// TwinCAT 3 PLC project PLC
// Title: AUT_Utilities
// Company: AU-tomation
// Author: Ing. Alberto Utili
// ProjectVersion: 1.0.0.0
// Description: AU-tomation Toolkit Utilities Library
// ProgramVersion: 3.1.4026.20
// libraries:
//   Tc2_Standard, * (Beckhoff Automation GmbH)
//   Tc2_System, * (Beckhoff Automation GmbH)
//   Tc2_Utilities, * (Beckhoff Automation GmbH)
//   Tc3_Module, * (Beckhoff Automation GmbH)
// project tree:
//   POUs/StringBuilder/Classes/ StringBuilder.TcPOU
//   POUs/StringBuilder/Interfaces/ ILimitedStringBuilder.TcIO, IStringBuilder.TcIO (not stored)
//   Project Information/ F_GetCompany.TcPOU, F_GetTitle.TcPOU, F_GetVersion.TcPOU
//   Version/ Global_Version.TcGVL

// ---- Version/Global_Version.TcGVL
{attribute 'TcGenerated'}
{attribute 'no-analysis'}
{attribute 'linkalways'}
// This function has been automatically generated from the project information.
VAR_GLOBAL CONSTANT
	{attribute 'const_non_replaced'}
	stLibVersion_AUT_Utilities : ST_LibVersion := (iMajor := 1, iMinor := 0, iBuild := 0, iRevision := 0, nFlags := 0, sVersion := '1.0.0.0');
END_VAR

// ---- POUs/StringBuilder/Interfaces/ILimitedStringBuilder.TcIO
INTERFACE ILimitedStringBuilder

METHOD  Append : IStringBuilder // Append text to t current build string.
VAR_INPUT
	Text : STRING(1024); //Text to append to current build string
END_VAR
END_METHOD

METHOD Reset : ILimitedStringBuilder //Reset current build string to an empty string.
END_METHOD

METHOD ToString : STRING(2048)    //Returns current build string.
END_METHOD

METHOD ToWString : WSTRING(2048) //Returns current build string.
END_METHOD

END_INTERFACE

// ---- POUs/StringBuilder/Classes/StringBuilder.TcPOU
FUNCTION_BLOCK PUBLIC StringBuilder IMPLEMENTS  IStringBuilder, ILimitedStringBuilder
VAR
	{attribute 'hide'}
	_BuildingString : STRING(2048);
END_VAR

METHOD PUBLIC Append : IStringBuilder // Append text to t current build string.
VAR_INPUT
	Text : STRING(1024); //Text to append to current build string
END_VAR
VAR
    _BoolRes : BOOL;
END_VAR
_BoolRes := Tc2_Utilities.CONCAT2(ADR(_BuildingString), ADR(Text), ADR(_BuildingString), SIZEOF(_BuildingString));
Append := THIS^;    // Fluent interface
END_METHOD

METHOD AssignDelimitedSubstringTo : IStringBuilder
VAR_INPUT
    Delimiter : STRING(1);
    SubstringIndex : UDINT;
	Destination : POINTER TO STRING(2048);
    DestinationSize : UDINT;
END_VAR
VAR
    _CurrentPosition : UDINT := 0;
    _CurrentDelimiterPosition : UDINT := 0;
    _CurrentDelimiterIndex : UDINT := 0;
    _LeadingDelimiterPosition : UDINT := 0;
    _TrailingDelimiterPosition : UDINT := 0;
    _Substring : STRING(2048) := '';
    _Index : UDINT;
    _BoolRes : BOOL;
END_VAR
// FOR _Index := 1 TO (SubstringIndex - 1) DO
//     _LeadingDelimiterPosition := Tc2_Utilities.FIND2(ADR(_BuildingString), ADR(Delimiter))
//     
// END_FOR

// ATTENTION: pointer arithmetics is used to move inside string
IF SubstringIndex < 1 THEN
    SubstringIndex := 1;
END_IF
REPEAT
    _CurrentDelimiterPosition := Tc2_Utilities.FIND2(ADR(_BuildingString) + _CurrentPosition, ADR(Delimiter));
    IF _CurrentDelimiterPosition > 0 THEN
        _CurrentPosition := _CurrentPosition + _CurrentDelimiterPosition;
        _CurrentDelimiterIndex := _CurrentDelimiterIndex + 1;
        IF _CurrentDelimiterIndex = (SubstringIndex - 1) THEN
            _LeadingDelimiterPosition := _CurrentPosition;
        END_IF
        IF _CurrentDelimiterIndex = SubstringIndex THEN
            _TrailingDelimiterPosition := _CurrentPosition;
        END_IF
    END_IF
    UNTIL _CurrentDelimiterPosition = 0 OR _CurrentDelimiterIndex = SubstringIndex
END_REPEAT

IF _CurrentDelimiterIndex = 0 THEN
    // No delimiter was found: assign entire building string
    _BoolRes := Tc2_Utilities.STRNCPY(Destination, ADR(_BuildingString), DestinationSize);       
ELSIF SubstringIndex > (_CurrentDelimiterIndex + 1) THEN
    // Requested substring not found: assign an empty string
    _BoolRes := Tc2_Utilities.STRNCPY(Destination, ADR(_Substring), DestinationSize);       
ELSE
    // Delimiters were found: assign requested substring
    // NOTE: STRNCPY inserts a null terminator at the position of destination size (for copying n chars: destination size must be n + 1)
    IF SubstringIndex = 1 THEN
        _BoolRes := Tc2_Utilities.STRNCPY(ADR(_Substring), ADR(_BuildingString), _TrailingDelimiterPosition);   
    ELSE
        _BoolRes := Tc2_Utilities.STRNCPY(ADR(_Substring), ADR(_BuildingString) + _LeadingDelimiterPosition, _TrailingDelimiterPosition - _LeadingDelimiterPosition);
    END_IF
    //_Substring[_TrailingDelimiterPosition - _LeadingDelimiterPosition] := 0;    // Put Null terminator at the end of the substring
    _BoolRes := Tc2_Utilities.STRNCPY(Destination, ADR(_Substring), DestinationSize);   
END_IF
AssignDelimitedSubstringTo := THIS^;      // Fluent interface
END_METHOD

METHOD AssignTo : IStringBuilder
VAR_INPUT
	Destination : POINTER TO STRING(2048);
    DestinationSize : UDINT;
END_VAR
VAR
    _BoolRes : BOOL;
END_VAR
_BoolRes := Tc2_Utilities.STRNCPY(Destination, ADR(_BuildingString), DestinationSize);
AssignTo := THIS^;      // Fluent interface
END_METHOD

METHOD PUBLIC InsertAt : IStringBuilder
VAR_INPUT
	Text : STRING(1024);
	Position : UDINT;
END_VAR
VAR
    _BoolRes : BOOL;
END_VAR
_BoolRes := Tc2_Utilities.INSERT2(ADR(_BuildingString), ADR(Text), ADR(_BuildingString), SIZEOF(_BuildingString), Position);
InsertAt := THIS^;      // Fluent interface
END_METHOD

METHOD  Left : IStringBuilder // Append text to t current build string.
VAR_INPUT
	Length : UDINT;
END_VAR
VAR
    _BoolRes : BOOL;
END_VAR
_BoolRes := Tc2_Utilities.DELETE2(ADR(_BuildingString), ADR(_BuildingString), SIZEOF(_BuildingString), Tc2_Utilities.LEN2(ADR(_BuildingString)) - Length, Length + 1);
Left := THIS^;      // Fluent interface
END_METHOD

METHOD  Mid : IStringBuilder // Append text to t current build string.
VAR_INPUT
	Position : UDINT;
	Length : UDINT;
END_VAR
VAR
    _BoolRes : BOOL;
END_VAR
_BoolRes := Tc2_Utilities.DELETE2(ADR(_BuildingString), ADR(_BuildingString), SIZEOF(_BuildingString), Position - 1, 1);
_BoolRes := Tc2_Utilities.DELETE2(ADR(_BuildingString), ADR(_BuildingString), SIZEOF(_BuildingString), Tc2_Utilities.LEN2(ADR(_BuildingString)) - Length, Length + 1);
Mid := THIS^;      // Fluent interface
END_METHOD

METHOD  PadLeft : IStringBuilder // Append text to t current build string.
VAR_INPUT
    PaddingChar : STRING(1);
	TotalLength : UDINT;
END_VAR
VAR
    _Index : UDINT;
    _PaddingString : STRING(1024) := '';
    _BoolRes : BOOL;
END_VAR
IF Tc2_Utilities.LEN2(ADR(_BuildingString)) < TotalLength THEN
    FOR _Index := 1 TO (TotalLength - Tc2_Utilities.LEN2(ADR(_BuildingString))) DO
        InsertAt(PaddingChar, 1);
    END_FOR   
END_IF
PadLeft := THIS^;      // Fluent interface
END_METHOD

METHOD  PadRight : IStringBuilder // Append text to t current build string.
VAR_INPUT
    PaddingChar : STRING(1);
	TotalLength : UDINT;
END_VAR
VAR
    _Index : UDINT;
    _PaddingString : STRING(1024) := '';
    _BoolRes : BOOL;
END_VAR
IF Tc2_Utilities.LEN2(ADR(_BuildingString)) < TotalLength THEN
    FOR _Index := 1 TO (TotalLength - Tc2_Utilities.LEN2(ADR(_BuildingString))) DO
        Append(PaddingChar);
    END_FOR   
END_IF
PadRight := THIS^;      // Fluent interface
END_METHOD

METHOD RemoveAt : IStringBuilder
VAR_INPUT
	Position : UDINT;
    Length : UDINT;
END_VAR
VAR
    _BoolRes : BOOL;
END_VAR
_BoolRes := Tc2_Utilities.DELETE2(ADR(_BuildingString), ADR(_BuildingString), SIZEOF(_BuildingString), Length, Position);
RemoveAt := THIS^;      // Fluent interface
END_METHOD

METHOD ReplaceAt : IStringBuilder
VAR_INPUT
    Text : STRING(1024);
	Position : UDINT;
    Length : UDINT;
END_VAR
VAR
    _BoolRes : BOOL;
END_VAR
_BoolRes := Tc2_Utilities.REPLACE2(ADR(_BuildingString), ADR(Text), ADR(_BuildingString), SIZEOF(_BuildingString), Length, Position);
ReplaceAt := THIS^;      // Fluent interface
END_METHOD

METHOD PUBLIC Reset : ILimitedStringBuilder //Reset current build string to an empty string.
_BuildingString := '';
Reset := THIS^;     // Fluent interface
END_METHOD

METHOD  Right : IStringBuilder // Append text to t current build string.
VAR_INPUT
	Length : UDINT;
END_VAR
VAR
    _BoolRes : BOOL;
END_VAR
_BoolRes := Tc2_Utilities.DELETE2(ADR(_BuildingString), ADR(_BuildingString), SIZEOF(_BuildingString), Tc2_Utilities.LEN2(ADR(_BuildingString)) - Length, 1);
Right := THIS^;      // Fluent interface
END_METHOD

METHOD PUBLIC ToString : STRING(2048) //Returns current build string.
ToString := _BuildingString;
END_METHOD

METHOD ToWString : WSTRING(2048) //Returns current build string.
ToWString := Tc2_Utilities.CHAR_TO_WCHAR(_BuildingString);
END_METHOD

END_FUNCTION_BLOCK

// ---- Project Information/F_GetCompany.TcPOU
// This function has been automatically generated from the project information.
{attribute 'signature_flag' := '1073741824'}
{attribute 'TcGenerated'}
{attribute 'no-analysis'}
FUNCTION F_GetCompany : WSTRING
VAR_INPUT
	
END_VAR

F_GetCompany := "AU-tomation";

END_FUNCTION

// ---- Project Information/F_GetTitle.TcPOU
// This function has been automatically generated from the project information.
{attribute 'signature_flag' := '1073741824'}
{attribute 'TcGenerated'}
{attribute 'no-analysis'}
FUNCTION F_GetTitle : WSTRING
VAR_INPUT
	
END_VAR

F_GetTitle := "AUT_Utilities";

END_FUNCTION

// ---- Project Information/F_GetVersion.TcPOU
// This function has been automatically generated from the project information.
{attribute 'signature_flag' := '1073741824'}
{attribute 'TcGenerated'}
{attribute 'no-analysis'}
FUNCTION F_GetVersion : ST_LibVersion
VAR_INPUT
	
END_VAR

F_GetVersion.iMajor := 1;
F_GetVersion.iMinor := 0;
F_GetVersion.iBuild := 0;
F_GetVersion.iRevision := 0;
F_GetVersion.sVersion := '1.0.0.0';
F_GetVersion.nFlags := 0;

END_FUNCTION
